// TwinCAT 3 PLC project Name
// ProgramVersion: 3.1.4026.17
// CompilerDefines: VISU_USEPROPERTYINFO
// libraries:
//   CmpBitmapPool, * (System)
//   Tc2_Standard, * (Beckhoff Automation GmbH)
//   Tc2_System, * (Beckhoff Automation GmbH)
//   Tc2_Utilities, * (Beckhoff Automation GmbH)
//   TextListUtils, * (System)
//   VisuDialogs, * (System)
//   VisuSymbols, 4.5.0.0 (System)
// project tree:
//   DUTs/ DUT_AlarmInfo.TcDUT (not stored), DUT_ModelInfo.TcDUT, DUT_ProductData.TcDUT (not stored)
//   / GlobalTextList.TcGTLO, PlcTask.TcTTO (not stored), Visualization Manager.TcVMO (not stored)
//   GVLs/ GVL_HMI.TcGVL, GVL_Retain.TcGVL, GVL_Status.TcGVL (not stored)
//   POUs/70_Data/ DataShift.TcPOU
//   POUs/80_HMI/ HMI.TcPOU (not stored)
//   POUs/99_FB/ fbAlarm.TcPOU (not stored), ModelInfoEquals.TcPOU
//   POUs/ MAIN.TcPOU (not stored), Test.TcPOU (not stored)
//   VISUs/ ImagePool.TcIPO (not stored), TextList.TcTLO (not stored)
//   VISUs/03_SideFrame/ LowerBar.TcVIS (not stored), SideBar.TcVIS (not stored), UpperBar.TcVIS (not stored)
//   VISUs/02_MainFrame/ Main.TcVIS (not stored), Data.TcVIS (not stored), Alarm.TcVIS (not stored), Setting.TcVIS (not stored), Manual.TcVIS (not stored), Model.TcVIS
//   VISUs/01_Page/ BasePage.TcVIS (not stored)
// real-time tasks:
//   TASK PlcTask: cycle T#10ms, priority 21, ADS port 351

// ---- DUTs/DUT_ModelInfo.TcDUT
TYPE DUT_ModelInfo :
STRUCT
	sName		: STRING;
	abType		: ARRAY[0..cMaxTypeNo-1] OF BOOL;
	aiType		: ARRAY[0..cMaxTypeNo-1] OF INT;
	arPosition	: ARRAY[0..cMaxAxisNo-1] OF LREAL;
	arSpeed		: ARRAY[0..cMaxAxisNo-1] OF LREAL;
END_STRUCT
END_TYPE

// ---- GVLs/GVL_HMI.TcGVL
//{attribute 'qualified_only'}
VAR_GLOBAL
	
	iSelectProductNo	: UINT; // Select Product No.
	bSaveProductData	: BOOL;
	bDeleteProductData	: BOOL;
	iSelectRecipeNo		: UINT;
	bSaveRecipeData		: BOOL;
	bDeleteRecipeData	: BOOL;
	bRemoveProductData	: BOOL;
	sCurrentTime		: STRING;
	
// Button
	bBtAutoMode			: BOOL;
	bBtStart			: BOOL;
	bBtStop				: BOOL;
	bBtHome				: BOOL;
	bBtDoorLock			: BOOL;
	bBtDoorUnlock		: BOOL;
	bBtAlarmReset		: BOOL;

// Lamp
	bLpBlink			: BOOL;
	bLpHome				: BOOL;
	bLpAlarmReset		: BOOL;
	bLpAutoMode			: BOOL;
	bLpStart			: BOOL;
	
// Index
	iTextIndex			: INT;	// By 'TextList' 0= Manual, 1= Auto
	iMainFrame			: INT; // 0= Main, 1= Manual, 2= Setting, 3= Model, 4= Data, 5= Alarm
	iModelIndex			: INT;

// Frame Number
    bMainScreen			: BOOL;
    bManualScreen		: BOOL;
	bSettingScreen		: BOOL;
	bModelScreen		: BOOL;
	bDataScreen			: BOOL;
	bAlarmScreen		: BOOL;
	
// Message Box
	sCurrentTitle		: STRING;
	sCurrentMessage		: STRING;
	bCallMessageBox		: BOOL;

// Time
	abStartTimeStamp	: ARRAY[0..cMaxStationNo-1] OF BOOL;
	abEndTimeStamp		: ARRAY[0..cMaxStationNo-1] OF BOOL;

// Test Bt
	bTest				: BOOL;
END_VAR

// ---- GVLs/GVL_Retain.TcGVL
//{attribute 'qualified_only'}
  {attribute 'TcPersistent'}
VAR_GLOBAL
//Product Data
	astProductData 		: ARRAY[0..cMaxStationNo+1] OF DUT_ProductData;
	abMoveShift			: ARRAY[0..cMaxStationNo] OF BOOL;

// Alarm
	astAlarmHistory		: ARRAY[0..cMaxAlarmLogCount-1] OF DUT_AlarmInfo; // 최근 100개 알람 저장

// Model
	astModel			: ARRAY[0..cMaxModelNo-1] OF dut_ModelInfo;
	astModelHmi			: ARRAY[0..cMaxModelNo-1] OF dut_ModelInfo;
	
END_VAR

VAR_GLOBAL CONSTANT
	cMaxAlarmLogCount	: INT := 100; 
	cMaxStationNo 		: INT := 30;
	cMaxTypeNo			: INT := 20;
	cMaxAxisNo			: INT := 30;
	cMaxModelNo			: INT := 10;
END_VAR

// ---- POUs/70_Data/DataShift.TcPOU
PROGRAM DataShift
VAR
	i					:INT; //loop index
END_VAR

// Local Time
	GVL_Status.fbLocalTime(bEnable := TRUE);	// Current Time

//Remove Total Product Data
	IF GVL_HMI.bRemoveProductData THEN
		FOR i := 0 TO cMaxStationNo DO
			astProductData[i] := astProductData[cMaxStationNo+1];
		END_FOR;
		GVL_HMI.bRemoveProductData := FALSE;
	END_IF

//Data Shift
	FOR i := 0 TO (cMaxStationNo) DO
		IF i > 0 AND i <= cMaxStationNo THEN  // 범위 체크 추가
			IF abMoveShift[i] = TRUE THEN
				astProductData[i] := astProductData[i-1];
				astProductData[i-1] := astProductData[cMaxStationNo+1]; // Delete Data before Station
				abMoveShift[i] := FALSE;
			END_IF
			
			IF abStartTimeStamp[i] AND GVL_Status.fbLocalTime.bValid THEN
				astProductData[i].dtStartTime := SYSTEMTIME_TO_DT(GVL_Status.fbLocalTime.systemTime);
			END_IF
			IF abEndTimeStamp[i] AND GVL_Status.fbLocalTime.bValid THEN
				astProductData[i].dtEndTime := SYSTEMTIME_TO_DT(GVL_Status.fbLocalTime.systemTime);
			END_IF		
			astProductData[i].tProcessTime	:= astProductData[i].dtEndTime - astProductData[i].dtStartTime;
		END_IF
	END_FOR;

END_PROGRAM

// ---- POUs/99_FB/ModelInfoEquals.TcPOU
FUNCTION ModelInfoEquals : BOOL
VAR_INPUT
    a : DUT_ModelInfo;
    b : DUT_ModelInfo;
END_VAR
VAR
    i : INT;
END_VAR


ModelInfoEquals := TRUE;
IF a.sName <> b.sName THEN
    ModelInfoEquals := FALSE;
END_IF
FOR i := 0 TO cMaxTypeNo - 1 DO
    IF a.abType[i] <> b.abType[i] THEN
        ModelInfoEquals := FALSE;
    END_IF
    IF a.aiType[i] <> b.aiType[i] THEN
        ModelInfoEquals := FALSE;
    END_IF
END_FOR
FOR i := 0 TO cMaxAxisNo - 1 DO
    IF a.arPosition[i] <> b.arPosition[i] THEN
        ModelInfoEquals := FALSE;
    END_IF
    IF a.arSpeed[i] <> b.arSpeed[i] THEN
        ModelInfoEquals := FALSE;
    END_IF
END_FOR

END_FUNCTION

// ---- GlobalTextList.TcGTLO
TEXTLIST GlobalTextList
  422 = '%.19s' | Korea: '%.19s' | English: '%.19s'
  75 = '%s'
  410 = 'a'
  851 = 'Active'
  609 = 'Alarm'
  662 = 'Alarm Code'
  947 = 'Alarm Page'
  35 = 'Alarm Reset'
  411 = 'AlarmCode'
  22 = 'AlarmMessage'
  147 = 'AlarmReset' | Korea: '초기화'
  23 = 'Alarm_Log'
  557 = 'Arkplus' | Korea: '화면인터페이스' | English: 'Standard_HMI'
  491 = 'Auto Mode'
  808 = 'AutoMode'
  787 = 'b'
  699 = 'Code'
  709 = 'Conveyor'
  122 = 'Data'
  161 = 'Data Page'
  226 = 'Door'
  850 = 'Door Close'
  103 = 'Door Open'
  567 = 'DoorClose'
  271 = 'English' | Korea: '영어' | English: 'English'
  697 = 'fdsafdafsda'
  217 = 'GroupBox'
  279 = 'Home'
  332 = 'Korea' | Korea: '한국어' | English: 'Korea'
  0 = 'Location'
  956 = 'Main'
  707 = 'Main Page'
  301 = 'Manual'
  775 = 'Manual Page'
  83 = 'ManualMode'
  186 = 'Message'
  376 = 'Model'
  313 = 'Model Page'
  136 = 'Name'
  536 = 'Parameter'
  403 = 'Priority'
  529 = 'Robot'
  204 = 'SafetyBypass'
  331 = 'Sample'
  239 = 'Setting'
  394 = 'Setting Page'
  125 = 'Speed'
  849 = 'Standard_HMI' | Korea: '화면인터페이스'
  261 = 'Start'
  606 = 'Stop'
  904 = 'Test'
  272 = 'Time Stamp'
  199 = 'TimeStamp'
  396 = 'TurnTable'
  712 = 'type'
  171 = 'yyyy‑MM‑dd\xa0HH:mm:ss'
END_TEXTLIST

// ---- VISUs/02_MainFrame/Model.TcVIS
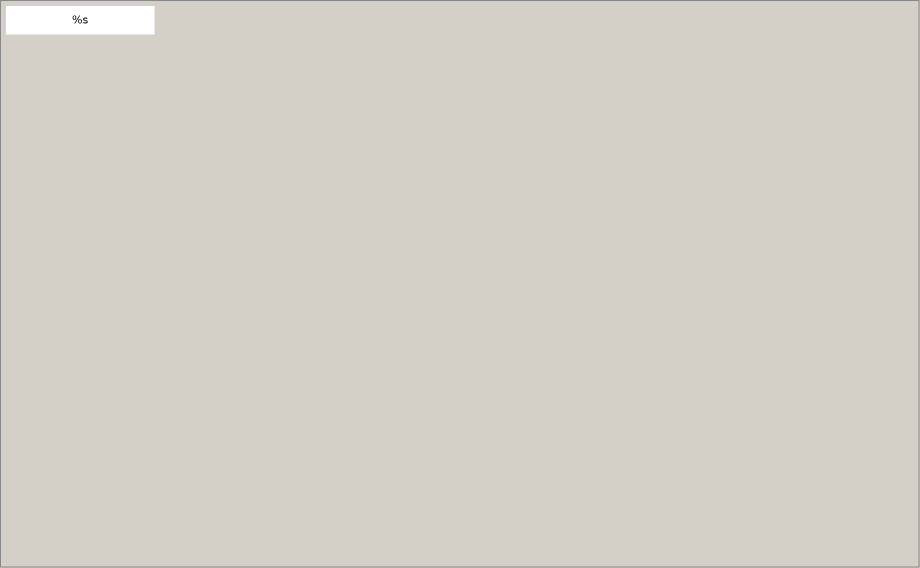
VISUALIZATION Model  // 920x568
    Textfield (5,5 150x30), "%s", text variable: astModel[iModelIndex].sName
END_VISUALIZATION
